FUNCTION_BLOCK Keypad
VAR_INPUT
	keyIn : ARRAY[0..7] OF BOOL;
	KeypadType: INT; 		//	0: tap switch | 1: toggle switch
END_VAR
VAR_OUTPUT
	keyOut : ARRAY[0..7] OF BOOL;
END_VAR
VAR
END_VAR


CASE KeypadType OF
	0:
		
	1:
ELSE
	;
END_CASE

END_FUNCTION_BLOCK

(* stored: Version 1.1.0.1, ProductVersion 3.1.4024.13
   POU Keypad: Id {d9e2ad64-99a7-4404-80a9-c6bcdb8547c7}, SpecialFunc None *)
